// TIA Portal V17 export
// export: Created 2025-03-10T12:19:18.9883578Z, ExportSetting WithDefaults, DisplayName Totally Integrated Automation Portal, DisplayVersion V17 Update 8, DisplayName TIA Portal Openness, DisplayVersion V17 Update 8, DisplayName TIA Portal Version Control Interface, DisplayVersion V17, DisplayName SINAMICS Startdrive Advanced, DisplayVersion V17 SP2, DisplayName SINAMICS Startdrive G110M, G120, G120C, G120D, G120P, G115D, DisplayVersion V17 SP2, DisplayName SINAMICS Startdrive G130, G150, S120, S150, SINAMICS MV, S210, DisplayVersion V17 SP2, DisplayName STEP 7 Professional, DisplayVersion V17 Update 8, DisplayName SINUMERIK ONE STEP 7 Toolbox, DisplayVersion V17 Update 12, DisplayName SINUMERIK 840D sl STEP 7 Toolbox, DisplayVersion V17 Update 12, DisplayName STEP 7 Safety, DisplayVersion V17 Update 6, DisplayName WinCC Advanced, DisplayVersion V17 Update 8
VAR_GLOBAL   // PLC tag table "TAGS_IO_SERVICES_CLADDING"
   "/////_COOLING_CHILLER_/////" AT %M8305.6 : Bool;   // /////_COOLING_CHILLER_/////
   "/////_OTHER_CIRCUIT_BREAKERS_/////" AT %M8308.0 : Bool;   // /////_OTHER_CIRCUIT_BREAKERS_/////
   "/////_OTHER_CONTACTOR_/////" AT %M8309.5 : Bool;   // /////_OTHER_CONTACTOR_/////
END_VAR
